PROPERTY P_scFuse_fbxEnable : CtaSysConfig.ITF_DATATYPE
GET
END_GET
END_PROPERTY

PROPERTY P_scFuse_fbxInputMb : CtaSysConfig.ITF_DATATYPE
GET
END_GET
END_PROPERTY

PROPERTY P_scFuse_fbxDoesAlarm : CtaSysConfig.ITF_DATATYPE
GET
END_GET
END_PROPERTY

PROPERTY P_scMotorFuse_fbxInputMb : CtaSysConfig.ITF_DATATYPE
GET
END_GET
END_PROPERTY

PROPERTY P_scMotorFuse_fbxEnable : CtaSysConfig.ITF_DATATYPE
GET
END_GET
END_PROPERTY

PROPERTY P_scMotorFuse_fbxDoesAlarm : CtaSysConfig.ITF_DATATYPE
GET
END_GET
END_PROPERTY

PROPERTY P_scManual_fbxAlowManualOn : CtaSysConfig.ITF_DATATYPE
GET
END_GET
END_PROPERTY

PROPERTY P_scManual_fbuiManualState : CtaSysConfig.ITF_DATATYPE
GET
END_GET
END_PROPERTY

PROPERTY P_scManual_fbrManualOnY : CtaSysConfig.ITF_DATATYPE
GET
END_GET
END_PROPERTY

PROPERTY P_scInfluxDb_fbxEnable : CtaSysConfig.ITF_DATATYPE
GET
END_GET
END_PROPERTY

PROPERTY P_scData_fbudiOperationStarts : CtaSysConfig.ITF_DATATYPE
GET
END_GET
END_PROPERTY

PROPERTY P_scData_fbudiOperatingHours : CtaSysConfig.ITF_DATATYPE
GET
END_GET
END_PROPERTY

PROPERTY proRefToRonYDumper : REFERENCE TO CtaAppDumper.fbDumper
GET
END_GET
END_PROPERTY

{attribute 'hide'} 
PROPERTY INTERNAL proCountedError : INT
GET
END_GET
END_PROPERTY

{attribute 'hide'} 
PROPERTY INTERNAL proCountedInfo : INT
GET
END_GET
END_PROPERTY

{attribute 'hide'} 
PROPERTY INTERNAL proITF_REPORTMANAGER : CtaAppReport.ITF_REPORTMANAGER
GET
END_GET
END_PROPERTY

{attribute 'hide'} 
PROPERTY INTERNAL proCountedWarning : INT
GET
END_GET
END_PROPERTY

PROPERTY INTERNAL proGetDI_MotorHand : BOOL
GET
END_GET
END_PROPERTY

{attribute 'hide'} 
PROPERTY proNotShowDI_MotorHand : BOOL
GET
END_GET
END_PROPERTY

PROPERTY proHandModul_ITF : CtaSysIO.ITF_IO
GET
END_GET
END_PROPERTY

PROPERTY proNotShowAI_ActualValue : BOOL
GET
END_GET
END_PROPERTY

PROPERTY proGetAI_ActualValue : REAL
GET
END_GET
END_PROPERTY

PROPERTY proActualValue_ITF : CtaSysIO.ITF_IO
GET
END_GET
END_PROPERTY

{attribute 'hide'} 
PROPERTY proNotShowDI_NoError : BOOL
GET
END_GET
END_PROPERTY

PROPERTY INTERNAL proGetDI_NoError : BOOL
GET
END_GET
END_PROPERTY

PROPERTY proNoError_ITF : CtaSysIO.ITF_IO
GET
END_GET
END_PROPERTY

{attribute 'hide'} 
PROPERTY proNotShowDI_RevisionSwitchOk : BOOL
GET
END_GET
END_PROPERTY

PROPERTY INTERNAL proGetDI_RevisionSwitchOK : BOOL
GET
END_GET
END_PROPERTY

PROPERTY proRevisionSwitch_ITF : CtaSysIO.ITF_IO
GET
END_GET
END_PROPERTY

{attribute 'hide'} 
PROPERTY proNotShowDI_IsOn : BOOL
GET
END_GET
END_PROPERTY

PROPERTY INTERNAL proGetDI_IsOn : BOOL
GET
END_GET
END_PROPERTY

PROPERTY proIsOn_ITF : CtaSysIO.ITF_IO
GET
END_GET
END_PROPERTY

{attribute 'hide'} 
PROPERTY proNotShowDI_MotorFuseOk : BOOL
GET
END_GET
END_PROPERTY

PROPERTY INTERNAL proGetDI_MotorFuseOk : BOOL
GET
END_GET
END_PROPERTY

PROPERTY proMotorFuse_ITF : CtaSysIO.ITF_IO
GET
END_GET
END_PROPERTY

{attribute 'hide'} 
PROPERTY proNotShowDI_FuseOk : BOOL
GET
END_GET
END_PROPERTY

PROPERTY INTERNAL proGetDI_FuseOK : BOOL
GET
END_GET
END_PROPERTY

PROPERTY proFuse_ITF : CtaSysIO.ITF_IO
GET
END_GET
END_PROPERTY

{attribute 'hide'} 
PROPERTY proNotShowDI_Ready : BOOL
GET
END_GET
END_PROPERTY

PROPERTY INTERNAL proGetDI_IsReady : BOOL
GET
END_GET
END_PROPERTY

PROPERTY proReady_ITF : CtaSysIO.ITF_IO
GET
END_GET
END_PROPERTY

PROPERTY proOn_ITF : CtaSysIO.ITF_IO
GET
END_GET
END_PROPERTY

PROPERTY proOnY_ITF : CtaSysIO.ITF_IO
GET
END_GET
END_PROPERTY

PROPERTY proIsRegulatet : BOOL
GET
END_GET
END_PROPERTY

PROPERTY proIsHandOnOrOff : BOOL
GET
END_GET
END_PROPERTY

PROPERTY proRunAfterTimeAktive : BOOL
GET
END_GET
END_PROPERTY

PROPERTY proLeadTimeAktive : BOOL
GET
END_GET
END_PROPERTY

PROPERTY proIsReady : BOOL
GET
END_GET
END_PROPERTY

PROPERTY proAuto : BOOL
GET
END_GET
SET
END_SET
END_PROPERTY

PROPERTY proHandOn : BOOL
SET
END_SET
GET
END_GET
END_PROPERTY

PROPERTY proIsError : BOOL
GET
END_GET
END_PROPERTY

PROPERTY proIsWarning : BOOL
GET
END_GET
END_PROPERTY

PROPERTY proEn : BOOL
GET
END_GET
SET
END_SET
END_PROPERTY

PROPERTY proHardWareHandModulAktive : BOOL
GET
END_GET
END_PROPERTY

PROPERTY proIsEnabled : BOOL
GET
END_GET
END_PROPERTY

PROPERTY proMotorIsOn : BOOL
GET
END_GET
END_PROPERTY

PROPERTY proHandOff : BOOL
SET
END_SET
GET
END_GET
END_PROPERTY

PROPERTY proRevisionSwitchOk : BOOL
GET
END_GET
END_PROPERTY

PROPERTY proHandOnY : REAL
SET
END_SET
GET
END_GET
END_PROPERTY

{attribute 'monitoring' := 'variable'}
PROPERTY proLockDown : BOOL
GET
END_GET
END_PROPERTY

{attribute 'monitoring' := 'variable'}
PROPERTY proAvailable : BOOL
GET
END_GET
END_PROPERTY

{attribute 'monitoring' := 'variable'}
PROPERTY proAcknowlege : BOOL
GET
END_GET
END_PROPERTY

PROPERTY proIconNr : UINT
SET
END_SET
GET
END_GET
END_PROPERTY

END_INTERFACE

// 30 Program Organization Units/fbAntrieb_Collector
FUNCTION_BLOCK fbAntrieb_Collector IMPLEMENTS ITF_ANTRIEB_COLLECTOR
VAR_INPUT
END_VAR
VAR_OUTPUT
END_VAR
VAR
    ayAT_INTERFACE          : ARRAY[1..Parameter.iMaxAT] OF ITF_ANTRIEB;   
    ayAT_INTERFACE_SORTET   : ARRAY[1..Parameter.iMaxAT] OF ITF_ANTRIEB; 
    xIsSortet               : BOOL;
    diNext                  : DINT    := 1;
    diMin                   : DINT    := 1;
    diMax                   : DINT;
    diMaxSort               : DINT;
    xError                  : BOOL;
    xBufferError            : BOOL;
    diMissedBuffer          : DINT;
END_VAR

METHOD metRegistry : DINT
VAR_INPUT
    ITF_AT_IN   :   ITF_ANTRIEB;
END_VAR
VAR
    diArrayPos  :   DINT;
    diCount     :   DINT;
END_VAR
IF ITF_AT_IN <> 0 THEN
    diArrayPos := __XADD(ADR(diNext),1);
    IF diArrayPos <= Parameter.iMaxAT AND diArrayPos >= 1 THEN
        IF __QUERYINTERFACE(ITF_AT_IN,ayAT_INTERFACE[diArrayPos]) THEN
            metRegistry             := diArrayPos;
            GVL_ANTRIEB.xValidData       := TRUE;
            diCount    := __XADD(ADR(diMax),1);
        END_IF;
    ELSE
        IF diArrayPos > Parameter.iMaxAT THEN
            xBufferError := TRUE;
            diMissedBuffer := diArrayPos - Parameter.iMaxAT;
		END_IF;
        xError      := TRUE; 
        metRegistry := 0;
    END_IF;   
ELSE
    xError := TRUE; 
    metRegistry := 0;
END_IF;
END_METHOD

METHOD metSortArray
VAR_INPUT
    stSearch    :   STRING;
    uiSort      :   UINT;
END_VAR
VAR
    diFor1      :   DINT;
    diFor2      :   DINT;
    diFill      :   DINT;
    ITF_AT_Temp :   ITF_ANTRIEB;    
    iBigger     :   INT;
END_VAR
IF stSearch <> '' THEN
    diMaxSort   := 0;
    diFill      := LOWER_BOUND(ayAT_INTERFACE,1); 
    FOR diFor1 := LOWER_BOUND(ayAT_INTERFACE,1) TO UPPER_BOUND(ayAT_INTERFACE,1) DO
        IF ayAT_INTERFACE[diFor1] <> 0 THEN
            IF FIND(ayAT_INTERFACE[diFor1].proGetBMK,stSearch) <> 0 OR FIND(ayAT_INTERFACE[diFor1].proGetVendorDesignation,stSearch) <> 0 THEN
                ayAT_INTERFACE_SORTET[diFill] := ayAT_INTERFACE[diFor1];
                diFill      := diFill + 1; 
                diMaxSort   := diFill -1; 
            END_IF;
        END_IF;
	END_FOR;
ELSE
    ayAT_INTERFACE_SORTET := ayAT_INTERFACE;
    diMaxSort := diMax;
END_IF; 
// 1 = Sort BMK
IF uiSort = 1 THEN
    FOR diFor1 := LOWER_BOUND(ayAT_INTERFACE_SORTET,1) TO diMaxSort DO 
        FOR diFor2 := LOWER_BOUND(ayAT_INTERFACE_SORTET,1) TO diMaxSort -1 DO 
            IF ayAT_INTERFACE_SORTET[diFor2] <> 0 AND ayAT_INTERFACE_SORTET[diFor2 + 1] <> 0 THEN
                IF LEN(ayAT_INTERFACE_SORTET[diFor2].proGetBMK) > LEN(ayAT_INTERFACE_SORTET[diFor2 + 1].proGetBMK) THEN
                    ITF_AT_Temp                         := ayAT_INTERFACE_SORTET[diFor2];
                    ayAT_INTERFACE_SORTET[diFor2]       := ayAT_INTERFACE_SORTET[diFor2 + 1];
                    ayAT_INTERFACE_SORTET[diFor2 + 1]   := ITF_AT_Temp; 
                ELSIF LEN(ayAT_INTERFACE_SORTET[diFor2].proGetBMK) = LEN(ayAT_INTERFACE_SORTET[diFor2 + 1].proGetBMK) THEN
                    iBigger := fcGetBigerStringValue(ayAT_INTERFACE_SORTET[diFor2].proGetBMK,ayAT_INTERFACE_SORTET[diFor2 + 1].proGetBMK);
                    IF iBigger = 1 THEN
                        ITF_AT_Temp                         := ayAT_INTERFACE_SORTET[diFor2];
                        ayAT_INTERFACE_SORTET[diFor2]       := ayAT_INTERFACE_SORTET[diFor2 + 1];
                        ayAT_INTERFACE_SORTET[diFor2 + 1]   := ITF_AT_Temp;                                                
					END_IF;
				END_IF;
            END_IF;       
        END_FOR;      
    END_FOR;     
// 2 = Sort Vendor Name    
ELSIF uiSort = 2 THEN
    FOR diFor1 := LOWER_BOUND(ayAT_INTERFACE_SORTET,1) TO diMaxSort DO 
        FOR diFor2 := LOWER_BOUND(ayAT_INTERFACE_SORTET,1) TO diMaxSort -1 DO 
            IF ayAT_INTERFACE_SORTET[diFor2] <> 0 AND ayAT_INTERFACE_SORTET[diFor2 + 1] <> 0 THEN
                iBigger := fcGetBigerStringValue(ayAT_INTERFACE_SORTET[diFor2].proGetVendorDesignation,ayAT_INTERFACE_SORTET[diFor2 + 1].proGetVendorDesignation);
                IF iBigger = 1 THEN
                    ITF_AT_Temp                         := ayAT_INTERFACE_SORTET[diFor2];
                    ayAT_INTERFACE_SORTET[diFor2]       := ayAT_INTERFACE_SORTET[diFor2 + 1];
                    ayAT_INTERFACE_SORTET[diFor2 + 1]   := ITF_AT_Temp;                                            
                END_IF;
            END_IF;       
        END_FOR;      
    END_FOR;
// 3 & 4 = Sort State  
ELSIF uiSort = 3 OR uiSort = 4 THEN
    FOR diFor1 := LOWER_BOUND(ayAT_INTERFACE_SORTET,1) TO diMaxSort DO 
        FOR diFor2 := LOWER_BOUND(ayAT_INTERFACE_SORTET,1) TO diMaxSort -1 DO 
            IF ayAT_INTERFACE_SORTET[diFor2] <> 0 AND ayAT_INTERFACE_SORTET[diFor2 + 1] <> 0 THEN
                IF ayAT_INTERFACE_SORTET[diFor2].proIsError < ayAT_INTERFACE_SORTET[diFor2 + 1].proIsError THEN
                    ITF_AT_Temp                         := ayAT_INTERFACE_SORTET[diFor2];
                    ayAT_INTERFACE_SORTET[diFor2]       := ayAT_INTERFACE_SORTET[diFor2 + 1];
                    ayAT_INTERFACE_SORTET[diFor2 + 1]   := ITF_AT_Temp;    
                ELSIF NOT ayAT_INTERFACE_SORTET[diFor2].proIsError THEN
                    IF ayAT_INTERFACE_SORTET[diFor2].proIsWarning < ayAT_INTERFACE_SORTET[diFor2 + 1].proIsWarning THEN
                        ITF_AT_Temp                         := ayAT_INTERFACE_SORTET[diFor2];
                        ayAT_INTERFACE_SORTET[diFor2]       := ayAT_INTERFACE_SORTET[diFor2 + 1];
                        ayAT_INTERFACE_SORTET[diFor2 + 1]   := ITF_AT_Temp;    
                    ELSIF ayAT_INTERFACE_SORTET[diFor2].proIsEnabled < ayAT_INTERFACE_SORTET[diFor2 + 1].proIsEnabled THEN
                        ITF_AT_Temp                         := ayAT_INTERFACE_SORTET[diFor2];
                        ayAT_INTERFACE_SORTET[diFor2]       := ayAT_INTERFACE_SORTET[diFor2 + 1];
                        ayAT_INTERFACE_SORTET[diFor2 + 1]   := ITF_AT_Temp; 
                    ELSIF ayAT_INTERFACE_SORTET[diFor2].proIsWarning AND ayAT_INTERFACE_SORTET[diFor2 + 1].proIsWarning THEN
                        IF ayAT_INTERFACE_SORTET[diFor2].proRevisionSwitchOk > ayAT_INTERFACE_SORTET[diFor2 + 1].proRevisionSwitchOk THEN         
                            ITF_AT_Temp                         := ayAT_INTERFACE_SORTET[diFor2];
                            ayAT_INTERFACE_SORTET[diFor2]       := ayAT_INTERFACE_SORTET[diFor2 + 1];
                            ayAT_INTERFACE_SORTET[diFor2 + 1]   := ITF_AT_Temp; 
                        END_IF;       
                    END_IF;                                                       
                END_IF;
            END_IF;       
        END_FOR;      
    END_FOR;    
// 5 = Sort Starts   
ELSIF uiSort = 5 THEN
    FOR diFor1 := LOWER_BOUND(ayAT_INTERFACE_SORTET,1) TO diMaxSort DO 
        FOR diFor2 := LOWER_BOUND(ayAT_INTERFACE_SORTET,1) TO diMaxSort -1 DO 
            IF ayAT_INTERFACE_SORTET[diFor2] <> 0 AND ayAT_INTERFACE_SORTET[diFor2 + 1] <> 0 THEN
                IF ayAT_INTERFACE_SORTET[diFor2].proCountedStarts < ayAT_INTERFACE_SORTET[diFor2 + 1].proCountedStarts THEN
                    ITF_AT_Temp                         := ayAT_INTERFACE_SORTET[diFor2];
                    ayAT_INTERFACE_SORTET[diFor2]       := ayAT_INTERFACE_SORTET[diFor2 + 1];
                    ayAT_INTERFACE_SORTET[diFor2 + 1]   := ITF_AT_Temp;                                            
                END_IF;
            END_IF;       
        END_FOR;      
    END_FOR; 
// 6 = Sort Stunden   
ELSIF uiSort = 6 THEN
    FOR diFor1 := LOWER_BOUND(ayAT_INTERFACE_SORTET,1) TO diMaxSort DO 
        FOR diFor2 := LOWER_BOUND(ayAT_INTERFACE_SORTET,1) TO diMaxSort -1 DO 
            IF ayAT_INTERFACE_SORTET[diFor2] <> 0 AND ayAT_INTERFACE_SORTET[diFor2 + 1] <> 0 THEN
                IF ayAT_INTERFACE_SORTET[diFor2].proCountedHours < ayAT_INTERFACE_SORTET[diFor2 + 1].proCountedHours THEN
                    ITF_AT_Temp                         := ayAT_INTERFACE_SORTET[diFor2];
                    ayAT_INTERFACE_SORTET[diFor2]       := ayAT_INTERFACE_SORTET[diFor2 + 1];
                    ayAT_INTERFACE_SORTET[diFor2 + 1]   := ITF_AT_Temp;                                            
                END_IF;
            END_IF;       
        END_FOR;      
    END_FOR;   
// 7 = Sort On   
ELSIF uiSort = 7 THEN
    FOR diFor1 := LOWER_BOUND(ayAT_INTERFACE_SORTET,1) TO diMaxSort DO 
        FOR diFor2 := LOWER_BOUND(ayAT_INTERFACE_SORTET,1) TO diMaxSort -1 DO 
            IF ayAT_INTERFACE_SORTET[diFor2] <> 0 AND ayAT_INTERFACE_SORTET[diFor2 + 1] <> 0 THEN
                IF ayAT_INTERFACE_SORTET[diFor2].proOn < ayAT_INTERFACE_SORTET[diFor2 + 1].proOn THEN
                    ITF_AT_Temp                         := ayAT_INTERFACE_SORTET[diFor2];
                    ayAT_INTERFACE_SORTET[diFor2]       := ayAT_INTERFACE_SORTET[diFor2 + 1];
                    ayAT_INTERFACE_SORTET[diFor2 + 1]   := ITF_AT_Temp;                                            
                END_IF;
            END_IF;       
        END_FOR;      
    END_FOR;   
ELSE
    uiSort := 0;     
END_IF; 
IF uiSort = 0 AND stSearch = '' THEN
    xIsSortet := FALSE;  
ELSE
    xIsSortet := TRUE;  
END_IF
END_METHOD

PROPERTY proMin : INT
GET
proMin := 1;
END_GET
END_PROPERTY

PROPERTY proMax : UINT
GET
IF xIsSortet THEN
    proMax := LIMIT(0,TO_UINT(diMaxSort),65535);    
ELSE
    proMax := LIMIT(0,TO_UINT(diMax),65535);    
END_IF
END_GET
END_PROPERTY

PROPERTY proayAntriebTabelle : ARRAY[1..Parameter.iMaxAT] OF ITF_ANTRIEB_TABELLE_INFO
GET
VAR
    diFor   :   DINT;
END_VAR
IF xIsSortet THEN
    FOR diFor := LOWER_BOUND(proayAntriebTabelle,1) TO UPPER_BOUND(proayAntriebTabelle,1) DO
        __QUERYINTERFACE(ayAT_INTERFACE_SORTET[diFor],proayAntriebTabelle[diFor]);   
	END_FOR
ELSE
    FOR diFor := LOWER_BOUND(proayAntriebTabelle,1) TO UPPER_BOUND(proayAntriebTabelle,1) DO
        __QUERYINTERFACE(ayAT_INTERFACE[diFor],proayAntriebTabelle[diFor]);   
	END_FOR
END_IF;
END_GET
END_PROPERTY

PROPERTY proMissedBuffer : DINT
GET
proMissedBuffer := diMissedBuffer;
END_GET
END_PROPERTY

PROPERTY proBufferError : BOOL
GET
proBufferError := xBufferError;
END_GET
END_PROPERTY

PROPERTY proayAntrieb : ARRAY[1..Parameter.iMaxAT] OF ITF_ANTRIEB
GET
VAR
    diFor   :   DINT;
END_VAR
IF xIsSortet THEN
    proayAntrieb := ayAT_INTERFACE_SORTET;
ELSE
    proayAntrieb := ayAT_INTERFACE;
END_IF;
END_GET
END_PROPERTY

METHOD metGetAntriebITF : ITF_ANTRIEB
VAR_INPUT
    iPos    :   INT;
END_VAR
IF TO_DINT(iPos) >= LOWER_BOUND(ayAT_INTERFACE,1) AND TO_DINT(iPos) <= UPPER_BOUND(ayAT_INTERFACE,1) THEN
    IF xIsSortet THEN
        metGetAntriebITF := ayAT_INTERFACE_SORTET[iPos];       
    ELSE
        metGetAntriebITF := ayAT_INTERFACE[iPos];       
	END_IF   
END_IF
END_METHOD

END_FUNCTION_BLOCK

// 21 Interface/ITF_ANTRIEB_COLLECTOR
INTERFACE ITF_ANTRIEB_COLLECTOR

PROPERTY proBufferError : BOOL
GET
END_GET
END_PROPERTY

METHOD metGetAntriebITF : ITF_ANTRIEB
VAR_INPUT
    iPos    :   INT;
END_VAR
END_METHOD

PROPERTY proMissedBuffer : DINT
GET
END_GET
END_PROPERTY

PROPERTY proMin : INT
GET
END_GET
END_PROPERTY

PROPERTY proMax : UINT
GET
END_GET
END_PROPERTY

PROPERTY proayAntriebTabelle : ARRAY[1..Parameter.iMaxAT] OF ITF_ANTRIEB_TABELLE_INFO
GET
END_GET
END_PROPERTY

METHOD metSortArray
VAR_INPUT
    stSearch    :   STRING;
    uiSort      :   UINT;
END_VAR
END_METHOD

END_INTERFACE

// 30 Program Organization Units/fcGetBigerStringValue
FUNCTION fcGetBigerStringValue : INT
VAR_INPUT
    st1     :   STRING(255);
    st2     :   STRING(255);
END_VAR
VAR
    diFor: DINT;
    diMax: DINT;
END_VAR

IF LEN(st1) > LEN(st2) THEN
    diMax := LEN(st2); 
    fcGetBigerStringValue := 1;
ELSIF LEN(st1) < LEN(st2) THEN
    diMax := LEN(st1);
    fcGetBigerStringValue := 2;     
ELSE
    diMax := LEN(st1);    
END_IF;
FOR diFor := 0 TO  diMax DO
    IF st1[diFor] > st2[diFor] THEN
        fcGetBigerStringValue := 1;  
        EXIT; 
    ELSIF st1[diFor] < st2[diFor] THEN
        fcGetBigerStringValue := 2;  
        EXIT;
    END_IF;
END_FOR;

END_FUNCTION

// 30 Program Organization Units/fcCheckQuerryAndIconReturn
FUNCTION fcCheckQuerryAndIconReturn : BOOL
VAR_INPUT
	_ITF_IN			: 	ITF_ANTRIEB;
	_uiIconNr_IN	:	UINT;
END_VAR

IF __QUERYINTERFACE(_ITF_IN,_ITF_IN) THEN
	fcCheckQuerryAndIconReturn := TRUE;	
	_ITF_IN.proIconNr := _uiIconNr_IN;
ELSE
	fcCheckQuerryAndIconReturn :=  FALSE;
END_IF

END_FUNCTION

// 40 Visualizations/COLLECTOR/VIS_ANTRIEB_COLLECTOR
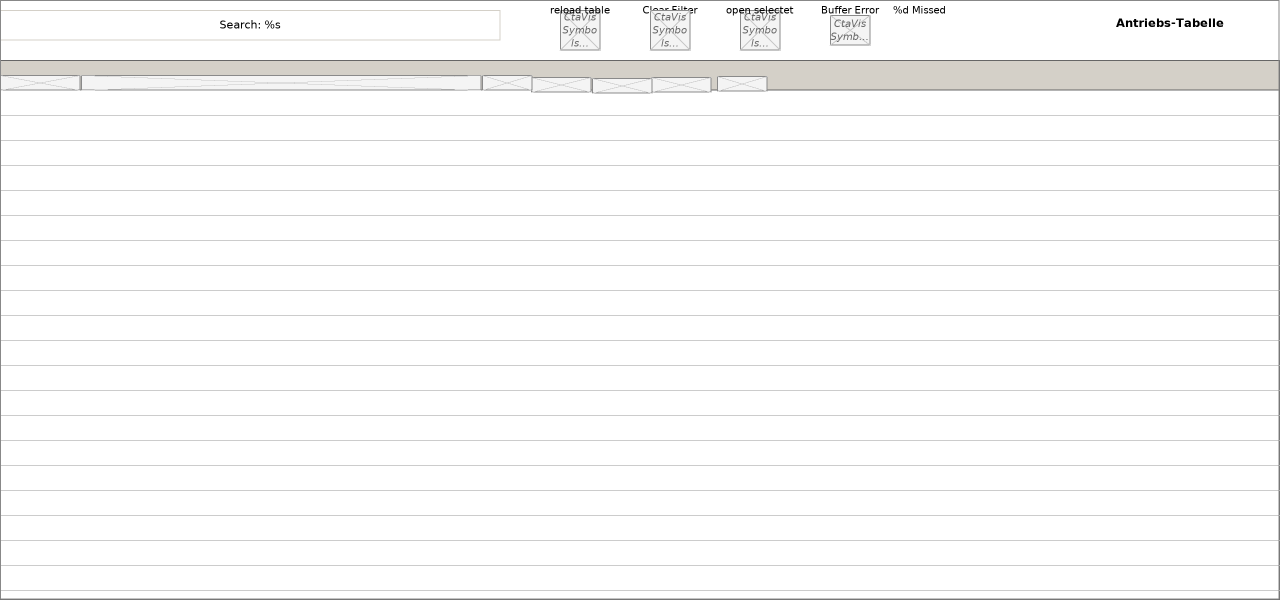
VISUALIZATION VIS_ANTRIEB_COLLECTOR  // 1280x600
    Frame (0,0 1280x600), invisible if: NOT GVL_ANTRIEB.xValidData
        shows VIS_ANTRIEB_COLLECTOR_TEMP(ayAntriebTabellenInfo := GVL_ANTRIEB.fbAntrieb_Collector.proayAntriebTabelle, uiMax := GVL_ANTRIEB.fbAntrieb_Collector.proMax, ITF_ANTRIEB_COLLECTOR := GVL_ANTRIEB.fbAntrieb_Collector)
END_VISUALIZATION

// 40 Visualizations/COLLECTOR/Help Funktionen/SelSort
VISUALIZATION SelSort  // 15x30
VAR_IN_OUT
	uiSel                       :   UINT;
END_VAR
VAR_INPUT
    stSearch                    :   STRING;    
    ITF_ANTRIEB_COLLECTOR       : ITF_ANTRIEB_COLLECTOR;
END_VAR
VAR_INPUT CONSTANT
    uiValue             :   UINT;
END_VAR
    Frame (0,15 15x15), invisible if: uiValue <> uiSel
        shows SortPfeil()
    Rectangle (0,0 15x30)
        OnMouseClick: execute {
            IF uiSel <> uiValue THEN
                uiSel   := uiValue;
            ELSE
                uiSel   := 0;
            END_IF
            ITF_ANTRIEB_COLLECTOR.metSortArray(stSearch,uiSel);
        }
END_VISUALIZATION

// 40 Visualizations/COLLECTOR/VIS_ANTRIEB_COLLECTOR_TEMP
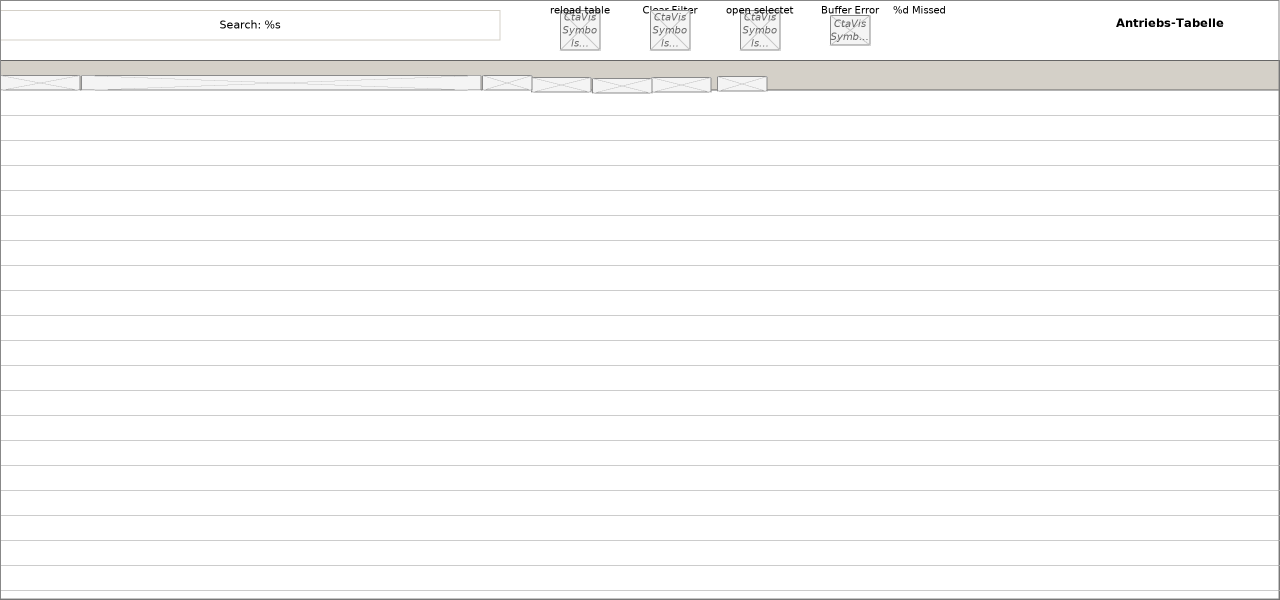
VISUALIZATION VIS_ANTRIEB_COLLECTOR_TEMP  // 1280x600
VAR_INPUT
	ayAntriebTabellenInfo   : ARRAY[1..Parameter.iMaxAT] OF ITF_ANTRIEB_TABELLE_INFO;
    uiMax                   : UINT;
    ITF_ANTRIEB_COLLECTOR   : ITF_ANTRIEB_COLLECTOR;
END_VAR
VAR
    iZeile                  :   INT;
    stSearch                :   STRING;
    uiSort                  :   UINT;
    xReadySearch            :   BOOL;
END_VAR
    Table (0,60 1280x540), data array: ayAntriebTabellenInfo
        p1128707560: uiMax
        p1014161805: Parameter.iMaxAT - 1 + 1
        p1137915858: iZeile
        p3726181087: ayAntriebTabellenInfo[INDEX].proNoBmkInList
        p3136911649: ayAntriebTabellenInfo[INDEX].proGetInstancePath
        p797552052: ayAntriebTabellenInfo[INDEX].proSetInstancePath
        p3854506369: ayAntriebTabellenInfo[INDEX].proGetBMK
        p1744040210: ayAntriebTabellenInfo[INDEX].proGetObjectId
        p290089404: ayAntriebTabellenInfo[INDEX].proGetCustomerDesignation
        p2319025000: ayAntriebTabellenInfo[INDEX].proGetAKS
        p511219082: Vendor designation
        p1892666644: ayAntriebTabellenInfo[INDEX].proGetVendorDesignation
        p4242324053: Run-on time
        p3863566920: ayAntriebTabellenInfo[INDEX].proRunAfterTime
        p1755163831: State
        p338671338: ayAntriebTabellenInfo[INDEX].proStateSymbol
        p505689113: Hours
        p1218418051: ayAntriebTabellenInfo[INDEX].proCountedHours
        p2340480326: ayAntriebTabellenInfo[INDEX].proBetriebsstunden
        p2237128397: Starts
        p3723444502: ayAntriebTabellenInfo[INDEX].proCountedStarts
        p4008173056: ayAntriebTabellenInfo[INDEX].proAnzahlStarts
        p4092479075: Enabled
        p2170511999: ayAntriebTabellenInfo[INDEX].proEnSymbol
        p4088588272: On IN
        p3104783080: ayAntriebTabellenInfo[INDEX].proIsOn
        p1757482276: On OUT
        p746581629: ayAntriebTabellenInfo[INDEX].proOn
        p1739542657: Lead time
        p1933151965: ayAntriebTabellenInfo[INDEX].proLeadTime
        p516019884: Y IN
        p7306298: ayAntriebTabellenInfo[INDEX].proIsOnY
        p2243050616: Y OUT
        p2501879983: ayAntriebTabellenInfo[INDEX].proOnY
    Image (740,10 40x40), invisible if: TO_DINT(iZeile) < LOWER_BOUND(ayAntriebTabellenInfo,1) OR TO_DINT(iZeile) > UPPER_BOUND(ayAntriebTabellenInfo,1), image: CtaVisSymbols.ImagePool.engine
        OnMouseClick:  Dialog=POPUP_ANTRIEB, Parameters={ITF_ANTRIEBIN: ITF_ANTRIEB_COLLECTOR.metGetAntriebITF(iZeile), uiPopUpGruppe: 0}, OpenModal=True, OpenCentered=True
    Textfield (0,10 500x30), "Search: %s", text variable: stSearch
        OnMouseClick: write the text variable via Default
        OnMouseClick: execute { xReadySearch := TRUE; }
    Image (560,10 40x40), invisible if: NOT xReadySearch, image: CtaVisSymbols.ImagePool.refresh_solo_black
        OnMouseClick: execute { ITF_ANTRIEB_COLLECTOR.metSortArray(stSearch,uiSort); xReadySearch := FALSE; }
    Label (540,5 80x10), "reload table", invisible if: NOT xReadySearch
    Label (720,5 80x10), "open selectet", invisible if: TO_DINT(iZeile) < LOWER_BOUND(ayAntriebTabellenInfo,1) OR TO_DINT(iZeile) > UPPER_BOUND(ayAntriebTabellenInfo,1)
    Label (630,5 80x10), "Clear Filter", invisible if: stSearch = '' AND uiSort = 0
    Image (650,10 40x40), invisible if: stSearch = '' AND uiSort = 0, image: CtaVisSymbols.ImagePool.close_solo_black
        OnMouseClick: execute {
            stSearch := '';
            uiSort   := 0;
            ITF_ANTRIEB_COLLECTOR.metSortArray(stSearch,uiSort);
            xReadySearch := FALSE;
        }
    Label (1095,8 150x30), "Antriebs-Tabelle"
    Label (810,5 80x10), "Buffer Error", invisible if: NOT ITF_ANTRIEB_COLLECTOR.proBufferError
    Image (830,15 40x30), invisible if: NOT ITF_ANTRIEB_COLLECTOR.proBufferError, image: CtaVisSymbols.ImagePool.CtaError
    Textfield (890,5 100x10), "%d Missed", text variable: ITF_ANTRIEB_COLLECTOR.proMissedBuffer, invisible if: NOT ITF_ANTRIEB_COLLECTOR.proBufferError
    Frame (717,61 50x30)
        shows SelSort(uiSel := uiSort, stSearch := stSearch, ITF_ANTRIEB_COLLECTOR := ITF_ANTRIEB_COLLECTOR, uiValue := 7)
    Frame (651,62 60x30)
        shows SelSort(uiSel := uiSort, stSearch := stSearch, ITF_ANTRIEB_COLLECTOR := ITF_ANTRIEB_COLLECTOR, uiValue := 6)
    Frame (592,63 60x30)
        shows SelSort(uiSel := uiSort, stSearch := stSearch, ITF_ANTRIEB_COLLECTOR := ITF_ANTRIEB_COLLECTOR, uiValue := 5)
    Frame (531,62 60x30)
        shows SelSort(uiSel := uiSort, stSearch := stSearch, ITF_ANTRIEB_COLLECTOR := ITF_ANTRIEB_COLLECTOR, uiValue := 4)
    Frame (482,60 50x30)
        shows SelSort(uiSel := uiSort, stSearch := stSearch, ITF_ANTRIEB_COLLECTOR := ITF_ANTRIEB_COLLECTOR, uiValue := 3)
    Frame (81,60 400x30)
        shows SelSort(uiSel := uiSort, stSearch := stSearch, ITF_ANTRIEB_COLLECTOR := ITF_ANTRIEB_COLLECTOR, uiValue := 2)
    Frame (0,60 80x30)
        shows SelSort(uiSel := uiSort, stSearch := stSearch, ITF_ANTRIEB_COLLECTOR := ITF_ANTRIEB_COLLECTOR, uiValue := 1)
END_VISUALIZATION

// 40 Visualizations/COLLECTOR/Help Funktionen/SortPfeil
VISUALIZATION SortPfeil  // 15x15
    Image (0,0 15x15), image: CtaVisSymbols.ImagePool.arrow-down_solo_black
END_VISUALIZATION

// 40 Visualizations/POPUP/POPUP_ANTRIEB
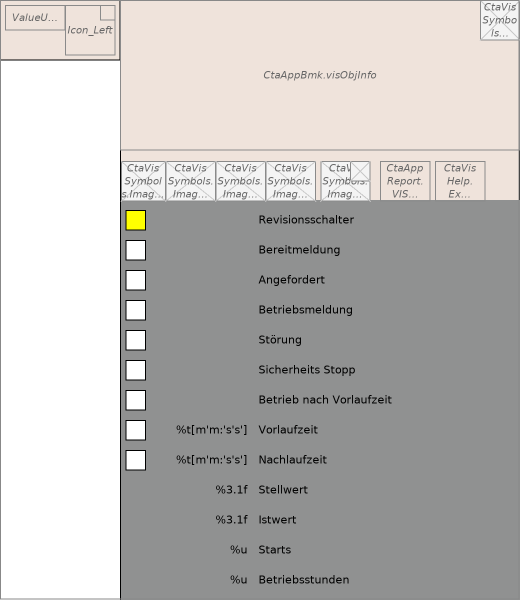
VISUALIZATION POPUP_ANTRIEB  // 520x600
VAR_INPUT
    ITF_ANTRIEBIN    	:   ITF_ANTRIEB;
	stExklParameter_IN	:	STRING[40];	
	uiPopUpGruppe 		: 	UINT;
END_VAR
    Rectangle (0,0 120x60)
    Rectangle (120,0 400x600)
    Frame (120,0 400x150)
        shows CtaAppBmk.visObjInfo(ITF_BMK_IN := ITF_ANTRIEBIN)
    Image (480,0 40x40), image: CtaVisSymbols.ImagePool.close_solo_black
        OnMouseClick:  Dialog=POPUP_ANTRIEB, Result=None, NumpadKeypadSet=True
    Frame (121,200 399x400), frame switch variable: uiPopUpGruppe
        shows VIS_ANTRIEB_OVERVIEW(ITF_ANTRIEBIN := ITF_ANTRIEBIN)
        shows VIS_ANTRIEB_MANUAL(ITF_ANTRIEBIN := ITF_ANTRIEBIN)
        shows VIS_ANTRIEB_PARAMETER(ITF_ANTRIEBIN := ITF_ANTRIEBIN)
        shows VIS_ANTRIEB_IO(ITF_ANTRIEBIN := ITF_ANTRIEBIN)
        shows AT_BUS(ITF_ANTRIEBIN := ITF_ANTRIEBIN)
        shows VIS_ANTRIEB_REPORTS(ITF_ANTRIEBIN := ITF_ANTRIEBIN)
        pReferences[2]: ITF_Parameter=ITF_ANTRIEBIN.proParameter
    Frame (121,161 399x40)
        shows VIS_ANTRIEB_LISTE(uiPopUpGruppe := uiPopUpGruppe, xHand := ITF_ANTRIEBIN.proIsHandOnOrOff, xHandOff := ITF_ANTRIEBIN.proHandOff, ITF_REPORTMANAGER_IN := ITF_ANTRIEBIN.proITF_REPORTMANAGER, xBusTestAktiv := ITF_ANTRIEBIN.proModbusTest, stExklParameter_IN := stExklParameter_IN)
    Frame (5,5 110x50), input disabled if: TRUE, frame switch variable: ITF_ANTRIEBIN.proIconNr
        shows VIS_ANTRIEB_LEFT_ABOVE(ITF_ANTRIEB_IN := ITF_ANTRIEBIN, stExklParameter := stExklParameter_IN)
        shows VIS_ANTRIEB_LEFT_BELOW(ITF_ANTRIEB_IN := ITF_ANTRIEBIN, stExklParameter := stExklParameter_IN)
        shows VIS_ANTRIEB_RIGHT_ABOVE(ITF_ANTRIEB_IN := ITF_ANTRIEBIN, stExklParameter := stExklParameter_IN)
        shows VIS_ANTRIEB_RIGHT_BELOW(ITF_ANTRIEB_IN := ITF_ANTRIEBIN, stExklParameter := stExklParameter_IN)
END_VISUALIZATION

// 40 Visualizations/POPUP/VIS_ANTRIEB_LISTE
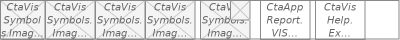
VISUALIZATION VIS_ANTRIEB_LISTE  // 400x40
VAR_IN_OUT
	uiPopUpGruppe 			:	UINT;
END_VAR
VAR_INPUT
    xHand           		: 	BOOL;
    xHandOff        		: 	BOOL;
    ITF_REPORTMANAGER_IN 	: 	CtaAppReport.ITF_REPORTMANAGER;
    xBusTestAktiv   		: 	BOOL;	
	stExklParameter_IN		:	STRING[40];
END_VAR
    Rectangle (100,0 40x40), colour toggle: uiPopUpGruppe = 2
        OnMouseDown: execute { uiPopUpGruppe := 2; }
    Rectangle (50,0 40x40), colour toggle: uiPopUpGruppe = 1
        OnMouseDown: execute { uiPopUpGruppe := 1; }
    Rectangle (0,0 40x40), colour toggle: uiPopUpGruppe = 0
        OnMouseDown: execute { uiPopUpGruppe := 0; }
    Image (0,0 45x40), image: CtaVisSymbols.ImagePool.eye
        OnMouseDown: execute { uiPopUpGruppe := 0; }
    Image (45,0 50x40), image: CtaVisSymbols.ImagePool.front_hand_Black
        OnMouseDown: execute { uiPopUpGruppe := 1; }
    Image (95,0 50x40), image: CtaVisSymbols.ImagePool.gear
        OnMouseDown: execute { uiPopUpGruppe := 2; }
    Image (45,0 50x40), invisible if: NOT xHand, image: CtaVisSymbols.ImagePool.front_hand_Yellow
        OnMouseDown: execute { uiPopUpGruppe := 1; }
    Rectangle (205,0 40x40), colour toggle: uiPopUpGruppe = 4
        OnMouseDown: execute { uiPopUpGruppe := 4; }
    Image (200,0 50x40), image: CtaVisSymbols.ImagePool.lan
        OnMouseDown: execute { uiPopUpGruppe := 4; }
    Image (45,0 50x40), invisible if: NOT xHandOff, image: CtaVisSymbols.ImagePool.front_hand_Yellow_Off
        OnMouseDown: execute { uiPopUpGruppe := 1; }
    Rectangle (150,0 40x40), colour toggle: uiPopUpGruppe = 3
        OnMouseDown: execute { uiPopUpGruppe := 3; }
    Image (145,0 50x40), image: CtaVisSymbols.ImagePool.dip-switch
        OnMouseDown: execute { uiPopUpGruppe := 3; }
    Image (230,0 20x20), invisible if: NOT xBusTestAktiv, image: CtaVisSymbols.ImagePool.front_hand_Yellow
        OnMouseDown: execute { uiPopUpGruppe := 4; }
    Rectangle (260,0 50x40), colour toggle: uiPopUpGruppe = 5
        OnMouseDown: execute { uiPopUpGruppe := 5; }
    Frame (260,0 50x40), input disabled if: TRUE
        shows CtaAppReport.VIS_ANZ_REPORTS_MODUL(ITF_REPORTMANAGER_IN := ITF_REPORTMANAGER_IN)
        OnMouseDown: execute { uiPopUpGruppe := 5; }
    Frame (315,0 50x40)
        shows CtaVisHelp.ExkParameterSymbol(stExklParameter := stExklParameter_IN)
END_VISUALIZATION

// 40 Visualizations/ICON/ANTRIEB_RIGHT/ANTRIEB_RIGHT_ABOVE/VIS_ANTRIEB_RigthAboveCheckQuerry
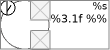
VISUALIZATION VIS_ANTRIEB_RigthAboveCheckQuerry  // 110x50
VAR_INPUT
    ITF_ANTRIEB_IN   :   ITF_ANTRIEB;	
END_VAR
VAR_INPUT
	stExklParameter		:	STRING[40];
END_VAR
    Frame (0,0 110x50)
        shows VIS_ANTRIEB_RigthAboveCheckIsEnabled(ITF_ANTRIEB_IN := ITF_ANTRIEB_IN, stExklParameter := stExklParameter)
END_VISUALIZATION

// 40 Visualizations/ICON/ANTRIEB_RIGHT/ANTRIEB_RIGHT_ABOVE/VIS_ANTRIEB_RIGHT_ABOVE
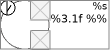
VISUALIZATION VIS_ANTRIEB_RIGHT_ABOVE  // 110x50
VAR_INPUT
    ITF_ANTRIEB_IN   :   ITF_ANTRIEB;	
END_VAR
VAR_INPUT CONSTANT
	stExklParameter		:	STRING[40] := ' ';
END_VAR
VAR CONSTANT
	uiIconNr		: UINT := 2;
END_VAR
    Frame (0,0 110x50), invisible if: NOT fcCheckQuerryAndIconReturn(_ITF_IN := ITF_ANTRIEB_IN, _uiIconNr_IN := uiIconNr)
        shows VIS_ANTRIEB_RigthAboveCheckQuerry(ITF_ANTRIEB_IN := ITF_ANTRIEB_IN, stExklParameter := stExklParameter)
END_VISUALIZATION

// 40 Visualizations/ICON/ANTRIEB_RIGHT/ANTRIEB_RIGHT_ABOVE/VIS_ANTRIEB_RigthAboveCheckIsEnabled
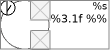
VISUALIZATION VIS_ANTRIEB_RigthAboveCheckIsEnabled  // 110x50
VAR_INPUT
    ITF_ANTRIEB_IN   :   ITF_ANTRIEB;	
END_VAR
VAR_INPUT
	stExklParameter		:	STRING[40];
END_VAR
    Frame (0,0 50x50), invisible if: NOT ITF_ANTRIEB_IN.proIsEnabled
        shows Icon_Right(ITF_ANTRIEB_IN := ITF_ANTRIEB_IN)
        shows Value_Right()
    Frame (50,0 60x25), invisible if: NOT ITF_ANTRIEB_IN.proIsEnabled
        shows ValueUpDwn(ITF_ANTRIEB_IN := ITF_ANTRIEB_IN, uiTextAusrichtung := 4)
    Frame (0,0 15x15), invisible if: NOT ITF_ANTRIEB_IN.proIsEnabled
        shows CommandOn(ITF_ANTRIEB_IN := ITF_ANTRIEB_IN)
    Rectangle (0,0 110x50)
        OnMouseClick:  Dialog=POPUP_ANTRIEB, Parameters={uiPopUpGruppe: 0, stExklParameter_IN: stExklParameter, ITF_ANTRIEBIN: ITF_ANTRIEB_IN}, OpenCentered=True
END_VISUALIZATION

// 40 Visualizations/ICON/ANTRIEB_BASE/CommandOn
VISUALIZATION CommandOn  // 15x15
VAR_INPUT
    ITF_ANTRIEB_IN   :   ITF_ANTRIEB;	
END_VAR
    Ellipse (0,0 15x15), colour toggle: ITF_ANTRIEB_IN.proOn
    Line (7,15) (7,10)
    Line (7,5) (7,0)
    Line (7,11) (11,5), invisible if: ITF_ANTRIEB_IN.proOn
    Line (7,15) (7,0), invisible if: NOT ITF_ANTRIEB_IN.proOn
END_VISUALIZATION

// 40 Visualizations/ICON/ANTRIEB_BASE/ICON/Icon_Left
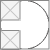
VISUALIZATION Icon_Left  // 50x50
VAR_INPUT
    ITF_ANTRIEB_IN   :   ITF_ANTRIEB;	
END_VAR
    Ellipse (0,0 49x49), colour toggle: ITF_ANTRIEB_IN.proMotorIsOn, invisible if: ITF_ANTRIEB_IN.proIsError
    Ellipse (0,0 49x49), colour toggle: ITF_ANTRIEB_IN.proIsError
    Image (0,0 20x20), invisible if: NOT ITF_ANTRIEB_IN.proIsWarning, image: CtaVisSymbols.ImagePool.CtaWarning
    Image (0,30 20x20), invisible if: NOT ITF_ANTRIEB_IN.proIsHandOnOrOff, image: CtaVisSymbols.ImagePool.front_hand_Yellow
    Image (0,30 20x20), invisible if: NOT ITF_ANTRIEB_IN.proHandOff, image: CtaVisSymbols.ImagePool.front_hand_Yellow_Off
END_VISUALIZATION

// 40 Visualizations/POPUP/PARAMETER/VIS_ANTRIEB_PARAMETER
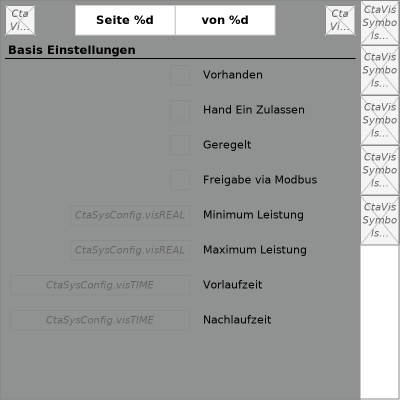
VISUALIZATION VIS_ANTRIEB_PARAMETER  // 400x400
VAR_INPUT
    ITF_ANTRIEBIN    :   ITF_ANTRIEB;	
END_VAR
VAR
    uiParameterGruppe : UINT;
END_VAR
    Image (145,122 150x30), image: ImagePool.Kreis
    Frame (360,0 40x300)
        shows VIS_ANTRIEB_PARAMETER_LISTE(uiParameterGruppe := uiParameterGruppe)
    Frame (0,0 360x400), frame switch variable: uiParameterGruppe
        shows VIS_ANTRIEB_PARAMETER_BASE(ITF_ANTRIEBIN := ITF_ANTRIEBIN)
        shows VIS_ANTRIEB_PARAMETER_FUSES(ITF_ANTRIEBIN := ITF_ANTRIEBIN)
        shows VIS_ANTRIEB_PARAMETER_IO(ITF_ANTRIEBIN := ITF_ANTRIEBIN)
        shows VIS_ANTRIEB_PARAMETER_DATA(ITF_ANTRIEBIN := ITF_ANTRIEBIN)
        shows VIS_ANTRIEB_PARAMETER_TRENDLOG(ITF_ANTRIEBIN := ITF_ANTRIEBIN)
        pReferences[0]: ITF_Parameter=ITF_Parameter
        pReferences[1]: ITF_Parameter=ITF_Parameter
        pReferences[2]: ITF_Parameter=ITF_Parameter
        pReferences[3]: ITF_Parameter=ITF_Parameter
        pReferences[4]: ITF_Parameter=ITF_Parameter
END_VISUALIZATION

// 40 Visualizations/POPUP/PARAMETER/VIS_ANTRIEB_PARAMETER_LISTE
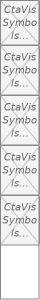
VISUALIZATION VIS_ANTRIEB_PARAMETER_LISTE  // 40x300
VAR_IN_OUT
	uiParameterGruppe : UINT;
END_VAR
    Rectangle (0,150 39x40), colour toggle: uiParameterGruppe = 3
        OnMouseDown: execute { uiParameterGruppe := 3; }
    Rectangle (0,100 39x40), colour toggle: uiParameterGruppe = 2
        OnMouseDown: execute { uiParameterGruppe := 2; }
    Rectangle (0,50 39x40), colour toggle: uiParameterGruppe = 1
        OnMouseDown: execute { uiParameterGruppe := 1; }
    Rectangle (0,0 39x40), colour toggle: uiParameterGruppe = 0
        OnMouseDown: execute { uiParameterGruppe := 0; }
    Image (0,0 40x45), image: CtaVisSymbols.ImagePool.engine
        OnMouseDown: execute { uiParameterGruppe := 0; }
    Image (0,45 40x50), image: CtaVisSymbols.ImagePool.lightning-bolt-circle
        OnMouseDown: execute { uiParameterGruppe := 1; }
    Image (0,95 40x50), image: CtaVisSymbols.ImagePool.dip-switch
        OnMouseDown: execute { uiParameterGruppe := 2; }
    Image (0,145 40x50), image: CtaVisSymbols.ImagePool.database_black
        OnMouseDown: execute { uiParameterGruppe := 3; }
    Rectangle (0,200 39x40), colour toggle: uiParameterGruppe = 4
        OnMouseDown: execute { uiParameterGruppe := 4; }
    Image (0,195 40x50), image: CtaVisSymbols.ImagePool.sine-wave
        OnMouseDown: execute { uiParameterGruppe := 4; }
END_VISUALIZATION

// 40 Visualizations/POPUP/MANUAL/VIS_ANTRIEB_MANUAL
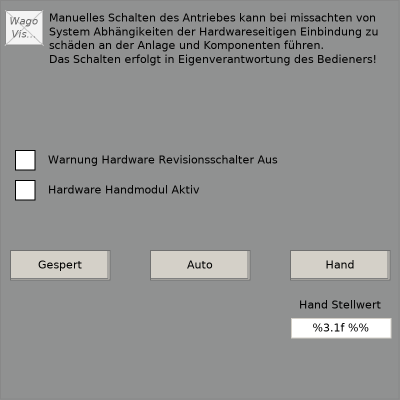
VISUALIZATION VIS_ANTRIEB_MANUAL  // 400x400
VAR_INPUT
    ITF_ANTRIEBIN    :   ITF_ANTRIEB;	
END_VAR
    Button (10,250 100x30), "Gespert", colour toggle: ITF_ANTRIEBIN.proHandOff, pressed state: ITF_ANTRIEBIN.proHandOff
        toggle ITF_ANTRIEBIN.proHandOff
    Button (290,250 100x30), "Hand", colour toggle: ITF_ANTRIEBIN.proHandOn, pressed state: ITF_ANTRIEBIN.proHandOn
        toggle ITF_ANTRIEBIN.proHandOn
    Button (150,250 100x30), "Auto", colour toggle: ITF_ANTRIEBIN.proAuto, pressed state: ITF_ANTRIEBIN.proAuto
        toggle ITF_ANTRIEBIN.proAuto
    Label (46,10 350x100), "Manuelles Schalten des Antriebes kann bei missachten von System Abhängikeiten der Hardwareseitigen Einbindung zu schäden an der Anlage und Komponenten führen. Das Schalten erfolgt in Eigenverantwortung des Bedieners!"
    Textfield (291,318 100x20), "%3.1f %%", text variable: ITF_ANTRIEBIN.proHandOnY, invisible if: NOT ITF_ANTRIEBIN.proIsRegulatet
        OnMouseClick: write the text variable via InputWithLimits, min 0, max 100, title 'Stellwert'
    Image (5,10 38x35), image: WagoVisuIcons.WagoIcons.2
    Label (290,295 100x20), "Hand Stellwert"
    Rectangle (15,180 20x20), colour toggle: ITF_ANTRIEBIN.proHardWareHandModulAktive, invisible if: NOT ITF_ANTRIEBIN.proHardWareHandModulAktive
    Label (45,180 200x20), "Hardware Handmodul Aktiv", invisible if: NOT ITF_ANTRIEBIN.proHardWareHandModulAktive
    Label (45,150 350x20), "Warnung Hardware Revisionsschalter Aus", invisible if: ITF_ANTRIEBIN.proRevisionSwitchOk
    Rectangle (15,150 20x20), colour toggle: NOT ITF_ANTRIEBIN.proRevisionSwitchOk, invisible if: ITF_ANTRIEBIN.proRevisionSwitchOk
END_VISUALIZATION

// 40 Visualizations/POPUP/OVERVIEW/VIS_ANTRIEB_OVERVIEW
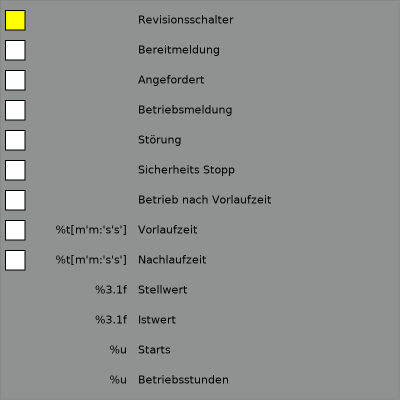
VISUALIZATION VIS_ANTRIEB_OVERVIEW  // 400x400
VAR_INPUT
    ITF_ANTRIEBIN    :   ITF_ANTRIEB;	
END_VAR
    Label (135,220 200x20), "Vorlaufzeit"
    Label (135,250 200x20), "Nachlaufzeit"
    Textfield (30,220 100x20), "%t[m'm:'s's']", text variable: ITF_ANTRIEBIN.proLeadTime
    Textfield (30,250 100x20), "%t[m'm:'s's']", text variable: ITF_ANTRIEBIN.proRunAfterTime
    Rectangle (5,220 20x20), colour toggle: ITF_ANTRIEBIN.proLeadTimeAktive
    Rectangle (5,250 20x20), colour toggle: ITF_ANTRIEBIN.proRunAfterTimeAktive
    Label (135,10 200x20), "Revisionsschalter"
    Label (135,40 200x20), "Bereitmeldung"
    Label (135,100 200x20), "Betriebsmeldung"
    Label (135,130 200x20), "Störung"
    Label (135,70 200x20), "Angefordert"
    Rectangle (5,10 20x20), colour toggle: ITF_ANTRIEBIN.proRevisionSwitchOk
    Rectangle (5,40 20x20), colour toggle: ITF_ANTRIEBIN.proIsReady
    Rectangle (5,70 20x20), colour toggle: ITF_ANTRIEBIN.proOn
    Rectangle (5,100 20x20), colour toggle: ITF_ANTRIEBIN.proMotorIsOn
    Rectangle (5,130 20x20), colour toggle: ITF_ANTRIEBIN.proIsError
    Label (135,160 200x20), "Sicherheits Stopp"
    Rectangle (5,160 20x20)
    Label (135,190 200x20), "Betrieb nach Vorlaufzeit"
    Rectangle (5,190 20x20), colour toggle: ITF_ANTRIEBIN.proIsOn
    Label (135,280 200x20), "Stellwert", invisible if: NOT ITF_ANTRIEBIN.proIsRegulatet
    Label (135,310 200x20), "Istwert", invisible if: NOT ITF_ANTRIEBIN.proIsRegulatet
    Textfield (30,280 100x20), "%3.1f", text variable: ITF_ANTRIEBIN.proOnY, invisible if: NOT ITF_ANTRIEBIN.proIsRegulatet
    Textfield (30,310 100x20), "%3.1f", text variable: ITF_ANTRIEBIN.proIsOnY, invisible if: NOT ITF_ANTRIEBIN.proIsRegulatet
    Textfield (30,370 100x20), "%u", text variable: ITF_ANTRIEBIN.proCountedHours
    Textfield (30,340 100x20), "%u", text variable: ITF_ANTRIEBIN.proCountedStarts
    Label (135,340 200x20), "Starts"
    Label (135,370 200x20), "Betriebsstunden"
END_VISUALIZATION

// 40 Visualizations/POPUP/BUS/AT_BUS
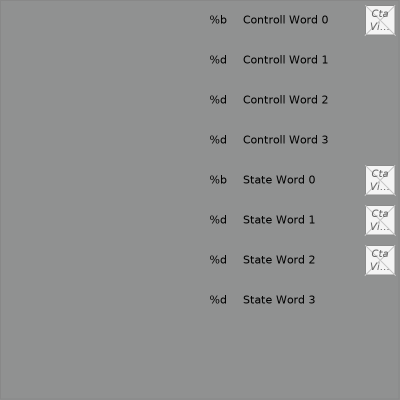
VISUALIZATION AT_BUS  // 400x400
VAR_INPUT
    ITF_ANTRIEBIN    :   ITF_ANTRIEB;	
END_VAR
    Frame (100,0 300x350)
        shows AT_BUS_CS(ITF_ANTRIEBIn := ITF_ANTRIEBIN, ayControllWord := ITF_ANTRIEBIN.proModbusControllWord, ayStateWord := ITF_ANTRIEBIN.proModbusStateWord)
END_VISUALIZATION

// 40 Visualizations/POPUP/BUS/AT_BUS_SW0_Detail
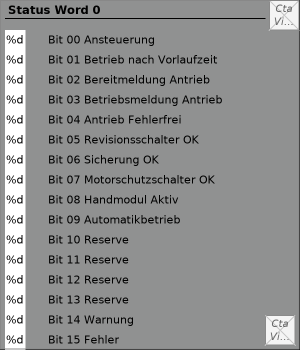
VISUALIZATION AT_BUS_SW0_Detail  // 300x350
VAR_IN_OUT
    wDetail     :   WORD;
END_VAR
VAR_INPUT	
    ITF_ANTRIEBIN    :   ITF_ANTRIEB;
END_VAR
VAR_IN_OUT
    xShow       :   BOOL;
END_VAR
    Rectangle (0,0 300x350)
    Textfield (5,30 20x20), "%d", text variable: TO_WORD(wDetail.0), input disabled if: NOT ITF_ANTRIEBIn.proModbusTest
        OnMouseClick: execute { wDetail.0 := NOT wDetail.0; }
    Label (45,30 220x20), "Bit 00 Ansteuerung"
    Textfield (5,50 20x20), "%d", text variable: TO_WORD(wDetail.1), input disabled if: NOT ITF_ANTRIEBIn.proModbusTest
        OnMouseClick: execute { wDetail.1 := NOT wDetail.1; }
    Label (45,50 220x20), "Bit 01 Betrieb nach Vorlaufzeit"
    Textfield (5,70 20x20), "%d", text variable: TO_WORD(wDetail.2), input disabled if: NOT ITF_ANTRIEBIn.proModbusTest
        OnMouseClick: execute { wDetail.2 := NOT wDetail.2; }
    Label (45,70 220x20), "Bit 02 Bereitmeldung Antrieb"
    Textfield (5,90 20x20), "%d", text variable: TO_WORD(wDetail.3), input disabled if: NOT ITF_ANTRIEBIn.proModbusTest
        OnMouseClick: execute { wDetail.3 := NOT wDetail.3; }
    Label (45,90 220x20), "Bit 03 Betriebsmeldung Antrieb"
    Textfield (5,110 20x20), "%d", text variable: TO_WORD(wDetail.4), input disabled if: NOT ITF_ANTRIEBIn.proModbusTest
        OnMouseClick: execute { wDetail.4 := NOT wDetail.4; }
    Label (45,110 220x20), "Bit 04 Antrieb Fehlerfrei"
    Textfield (5,130 20x20), "%d", text variable: TO_WORD(wDetail.5), input disabled if: NOT ITF_ANTRIEBIn.proModbusTest
        OnMouseClick: execute { wDetail.5 := NOT wDetail.5; }
    Label (45,130 220x20), "Bit 05 Revisionsschalter OK"
    Textfield (5,150 20x20), "%d", text variable: TO_WORD(wDetail.6), input disabled if: NOT ITF_ANTRIEBIn.proModbusTest
        OnMouseClick: execute { wDetail.6 := NOT wDetail.6; }
    Label (45,150 220x20), "Bit 06 Sicherung OK"
    Textfield (5,170 20x20), "%d", text variable: TO_WORD(wDetail.7), input disabled if: NOT ITF_ANTRIEBIn.proModbusTest
        OnMouseClick: execute { wDetail.7 := NOT wDetail.7; }
    Label (45,170 220x20), "Bit 07 Motorschutzschalter OK"
    Textfield (5,190 20x20), "%d", text variable: TO_WORD(wDetail.8), input disabled if: NOT ITF_ANTRIEBIn.proModbusTest
        OnMouseClick: execute { wDetail.8 := NOT wDetail.8; }
    Label (45,190 220x20), "Bit 08 Handmodul Aktiv"
    Textfield (5,210 20x20), "%d", text variable: TO_WORD(wDetail.9), input disabled if: NOT ITF_ANTRIEBIn.proModbusTest
        OnMouseClick: execute { wDetail.9 := NOT wDetail.9; }
    Label (45,210 220x20), "Bit 09 Automatikbetrieb"
    Textfield (5,230 20x20), "%d", text variable: TO_WORD(wDetail.10), input disabled if: NOT ITF_ANTRIEBIn.proModbusTest
        OnMouseClick: execute { wDetail.10 := NOT wDetail.10; }
    Label (45,230 220x20), "Bit 10 Reserve"
    Textfield (5,250 20x20), "%d", text variable: TO_WORD(wDetail.11), input disabled if: NOT ITF_ANTRIEBIn.proModbusTest
        OnMouseClick: execute { wDetail.11 := NOT wDetail.11; }
    Label (45,250 220x20), "Bit 11 Reserve"
    Textfield (5,270 20x20), "%d", text variable: TO_WORD(wDetail.12), input disabled if: NOT ITF_ANTRIEBIn.proModbusTest
        OnMouseClick: execute { wDetail.12 := NOT wDetail.12; }
    Label (45,270 220x20), "Bit 12 Reserve"
    Textfield (5,290 20x20), "%d", text variable: TO_WORD(wDetail.13), input disabled if: NOT ITF_ANTRIEBIn.proModbusTest
        OnMouseClick: execute { wDetail.13 := NOT wDetail.13; }
    Label (45,290 220x20), "Bit 13 Reserve"
    Textfield (5,310 20x20), "%d", text variable: TO_WORD(wDetail.14), input disabled if: NOT ITF_ANTRIEBIn.proModbusTest
        OnMouseClick: execute { wDetail.14 := NOT wDetail.14; }
    Label (45,310 220x20), "Bit 14 Warnung"
    Textfield (5,330 20x20), "%d", text variable: TO_WORD(wDetail.15), input disabled if: NOT ITF_ANTRIEBIn.proModbusTest
        OnMouseClick: execute { wDetail.15 := NOT wDetail.15; }
    Label (45,330 220x20), "Bit 15 Fehler"
    Image (269,0 30x30), image: CtaVisSymbols.ImagePool.close_solo_black
        OnMouseClick: execute { xShow := FALSE; ITF_ANTRIEBIN.proModbusTest := FALSE; }
    Label (5,0 150x20), "Status Word 0"
    Image (265,315 30x30), invisible if: ITF_ANTRIEBIN.proModbusTest, image: CtaVisSymbols.ImagePool.front_hand_Black
        OnMouseClick: execute { ITF_ANTRIEBIN.proModbusTest := TRUE; }
    Image (265,315 30x30), invisible if: NOT ITF_ANTRIEBIN.proModbusTest, image: CtaVisSymbols.ImagePool.front_hand_Yellow
        OnMouseClick: execute { ITF_ANTRIEBIN.proModbusTest := False; }
    Line (5,18) (265,18)
END_VISUALIZATION

// 40 Visualizations/POPUP/BUS/AT_BUS_CW0_Detail
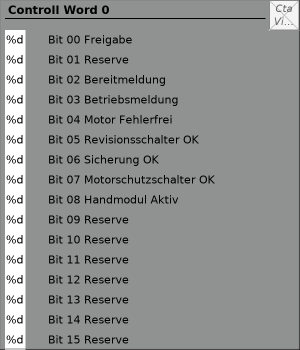
VISUALIZATION AT_BUS_CW0_Detail  // 300x350
VAR_IN_OUT
    wDetail :   WORD;
END_VAR
VAR_IN_OUT
    xShow   :   BOOL;
END_VAR
    Rectangle (0,0 300x350)
    Textfield (5,30 20x20), "%d", text variable: TO_WORD(wDetail.0), input disabled if: TRUE
    Label (45,30 180x20), "Bit 00 Freigabe"
    Textfield (5,50 20x20), "%d", text variable: TO_WORD(wDetail.1), input disabled if: TRUE
    Label (45,50 180x20), "Bit 01 Reserve"
    Textfield (5,70 20x20), "%d", text variable: TO_WORD(wDetail.2), input disabled if: TRUE
    Label (45,70 180x20), "Bit 02 Bereitmeldung"
    Textfield (5,90 20x20), "%d", text variable: TO_WORD(wDetail.3), input disabled if: TRUE
    Label (45,90 180x20), "Bit 03 Betriebsmeldung"
    Textfield (5,110 20x20), "%d", text variable: TO_WORD(wDetail.4), input disabled if: TRUE
    Label (45,110 180x20), "Bit 04 Motor Fehlerfrei"
    Textfield (5,130 20x20), "%d", text variable: TO_WORD(wDetail.5), input disabled if: TRUE
    Label (45,130 180x20), "Bit 05 Revisionsschalter OK"
    Textfield (5,150 20x20), "%d", text variable: TO_WORD(wDetail.6), input disabled if: TRUE
    Label (45,150 180x20), "Bit 06 Sicherung OK"
    Textfield (5,170 20x20), "%d", text variable: TO_WORD(wDetail.7), input disabled if: TRUE
    Label (45,170 180x20), "Bit 07 Motorschutzschalter OK"
    Textfield (5,190 20x20), "%d", text variable: TO_WORD(wDetail.8), input disabled if: TRUE
    Label (45,190 180x20), "Bit 08 Handmodul Aktiv"
    Textfield (5,210 20x20), "%d", text variable: TO_WORD(wDetail.9), input disabled if: TRUE
    Label (45,210 180x20), "Bit 09 Reserve"
    Textfield (5,230 20x20), "%d", text variable: TO_WORD(wDetail.10), input disabled if: TRUE
    Label (45,230 180x20), "Bit 10 Reserve"
    Textfield (5,250 20x20), "%d", text variable: TO_WORD(wDetail.11), input disabled if: TRUE
    Label (45,250 180x20), "Bit 11 Reserve"
    Textfield (5,270 20x20), "%d", text variable: TO_WORD(wDetail.12), input disabled if: TRUE
    Label (45,270 180x20), "Bit 12 Reserve"
    Textfield (5,290 20x20), "%d", text variable: TO_WORD(wDetail.13), input disabled if: TRUE
    Label (45,290 180x20), "Bit 13 Reserve"
    Textfield (5,310 20x20), "%d", text variable: TO_WORD(wDetail.14), input disabled if: TRUE
    Label (45,310 180x20), "Bit 14 Reserve"
    Textfield (5,330 20x20), "%d", text variable: TO_WORD(wDetail.15), input disabled if: TRUE
    Label (45,330 180x20), "Bit 15 Reserve"
    Image (269,0 30x30), image: CtaVisSymbols.ImagePool.close_solo_black
        OnMouseClick: execute { xShow := FALSE; }
    Label (5,0 150x20), "Controll Word 0"
    Line (5,18) (265,18)
END_VISUALIZATION

// 40 Visualizations/POPUP/BUS/AT_BUS_CS
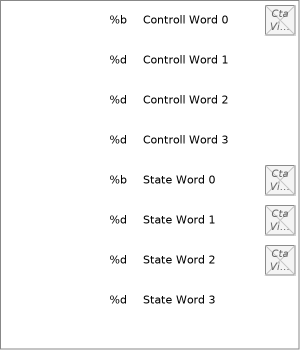
VISUALIZATION AT_BUS_CS  // 300x350
VAR_INPUT
    ITF_ANTRIEBIn        :   ITF_ANTRIEB;
    ayControllWord  :   REFERENCE TO ARRAY[0..3] OF WORD;
    ayStateWord     :   REFERENCE TO ARRAY[0..3] OF WORD;
END_VAR
VAR
    xShowCw :   BOOL;
    xShowSw :   BOOL;
    xShowSw1:   BOOL;
    xShowSw2:   BOOL;
END_VAR
    Textfield (0,10 130x20), "%b", text variable: ayControllWord[0]
    Label (140,10 120x20), "Controll Word 0"
    Label (140,50 120x20), "Controll Word 1"
    Textfield (0,50 130x20), "%d", text variable: ayControllWord[1]
    Label (140,90 120x20), "Controll Word 2", invisible if: TRUE
    Textfield (0,90 130x20), "%d", text variable: ayControllWord[2], invisible if: TRUE
    Label (140,130 120x20), "Controll Word 3", invisible if: TRUE
    Textfield (0,130 130x20), "%d", text variable: ayControllWord[2], invisible if: TRUE
    Image (265,5 30x30), image: CtaVisSymbols.ImagePool.information-variant
        OnMouseClick: execute {
            xShowCw := TRUE;
            xShowSw := FALSE;
            xShowSw1:= FALSE;
            xShowSw2:= FALSE;
        }
    Frame (300,0 300x350), invisible if: NOT xShowCw
        shows AT_BUS_CW0_Detail(wDetail := ayControllWord[0], xShow := xShowCw)
    Label (140,290 120x20), "State Word 3", invisible if: TRUE
    Textfield (0,170 130x20), "%b", text variable: ayStateWord[0]
        OnMouseDown: write the text variable via Default
    Label (140,170 120x20), "State Word 0"
    Label (140,210 120x20), "State Word 1"
    Textfield (0,210 130x20), "%d", text variable: ayStateWord[1]
    Label (140,250 120x20), "State Word 2"
    Textfield (0,250 130x20), "%d", text variable: ayStateWord[2]
    Textfield (0,290 130x20), "%d", text variable: ayStateWord[2], invisible if: TRUE
    Image (265,165 30x30), image: CtaVisSymbols.ImagePool.information-variant
        OnMouseClick: execute {
            xShowCw := FALSE;
            xShowSw := TRUE;
            xShowSw1:= FALSE;
            xShowSw2:= FALSE;
        }
    Frame (300,0 300x350), invisible if: NOT xShowSw
        shows AT_BUS_SW0_Detail(wDetail := ayStateWord[0], ITF_ANTRIEBIn := ITF_ANTRIEBIn, xShow := xShowSw)
        pReferences[0]: ITF_ATIn=ITF_ATIn
    Image (265,205 30x30), image: CtaVisSymbols.ImagePool.information-variant
        OnMouseClick: execute {
            xShowCw := FALSE;
            xShowSw := FALSE;
            xShowSw1:= TRUE;
            xShowSw2:= FALSE;
        }
    Frame (300,0 300x350), invisible if: NOT xShowSw1
        shows AT_BUS_SW1_Detail(wDetail := ayStateWord[1], ITF_ANTRIEBIn := ITF_ANTRIEBIn, xShow := xShowSw1)
    Frame (300,0 300x350), invisible if: NOT xShowSw2
        shows AT_BUS_SW2_Detail(wDetail := ayStateWord[2], ITF_ANTRIEBIn := ITF_ANTRIEBIn, xShow := xShowSw2)
    Image (265,245 30x30), image: CtaVisSymbols.ImagePool.information-variant
        OnMouseClick: execute {
            xShowCw := FALSE;
            xShowSw := FALSE;
            xShowSw1:= FALSE;
            xShowSw2:= TRUE;
        }
END_VISUALIZATION

// 40 Visualizations/POPUP/BUS/AT_BUS_SW1_Detail
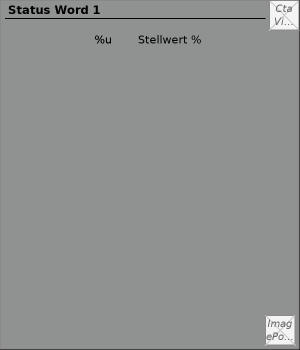
VISUALIZATION AT_BUS_SW1_Detail  // 300x350
VAR_IN_OUT
    wDetail     :   WORD;
END_VAR
VAR_INPUT	
    ITF_ANTRIEBIN    :   ITF_ANTRIEB;
END_VAR
VAR_IN_OUT
    xShow       :   BOOL;
END_VAR
    Rectangle (0,0 300x350)
    Image (269,0 30x30), image: CtaVisSymbols.ImagePool.close_solo_black
        OnMouseClick: execute { xShow := FALSE; ITF_ANTRIEBIN.proModbusTest := FALSE; }
    Label (5,0 150x20), "Status Word 1"
    Image (265,315 30x30), invisible if: ITF_ANTRIEBIN.proModbusTest, image: ImagePool.front_hand_FILL0_wght400_GRAD0_opsz48
        OnMouseClick: execute { ITF_ANTRIEBIN.proModbusTest := TRUE; }
    Image (265,315 30x30), invisible if: NOT ITF_ANTRIEBIn.proModbusTest, image: ImagePool.front_hand_FILL0_wght400_GRAD0_opsz48Yellow
        OnMouseClick: execute { ITF_ANTRIEBIN.proModbusTest := False; }
    Label (135,30 120x20), "Stellwert %"
    Textfield (5,30 110x20), "%u", text variable: wDetail, input disabled if: NOT ITF_ANTRIEBIn.proModbusTest
        OnMouseClick: write the text variable via InputWithLimits, min 0, max 100
    Textfield (5,30 110x20), "%u", text variable: wDetail, invisible if: ITF_ANTRIEBIN.proModbusTest
    Line (5,18) (265,18)
END_VISUALIZATION

// 40 Visualizations/POPUP/BUS/AT_BUS_SW2_Detail
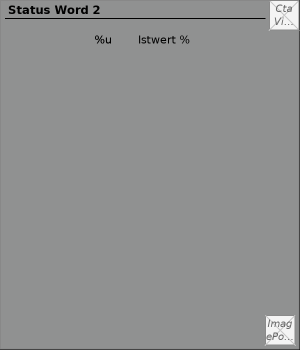
VISUALIZATION AT_BUS_SW2_Detail  // 300x350
VAR_IN_OUT
    wDetail             :   WORD;
END_VAR
VAR_INPUT	
    ITF_ANTRIEBIN       :   ITF_ANTRIEB;
END_VAR
VAR_IN_OUT
    xShow               :   BOOL;
END_VAR
    Rectangle (0,0 300x350)
    Image (269,0 30x30), image: CtaVisSymbols.ImagePool.close_solo_black
        OnMouseClick: execute { xShow := FALSE; ITF_ANTRIEBIN.proModbusTest := FALSE; }
    Label (5,0 150x20), "Status Word 2"
    Image (265,315 30x30), invisible if: ITF_ANTRIEBIn.proModbusTest, image: ImagePool.front_hand_FILL0_wght400_GRAD0_opsz48
        OnMouseClick: execute { ITF_ANTRIEBIN.proModbusTest := TRUE; }
    Image (265,315 30x30), invisible if: NOT ITF_ANTRIEBIN.proModbusTest, image: ImagePool.front_hand_FILL0_wght400_GRAD0_opsz48Yellow
        OnMouseClick: execute { ITF_ANTRIEBIN.proModbusTest := False; }
    Label (135,30 120x20), "Istwert %"
    Textfield (5,30 110x20), "%u", text variable: wDetail, input disabled if: NOT ITF_ANTRIEBIn.proModbusTest
        OnMouseClick: write the text variable via InputWithLimits, min 0, max 100
    Textfield (5,30 110x20), "%u", text variable: wDetail, invisible if: ITF_ANTRIEBIN.proModbusTest
    Line (5,18) (265,18)
END_VISUALIZATION

// 40 Visualizations/POPUP/REPORTS/VIS_ANTRIEB_REPORTS
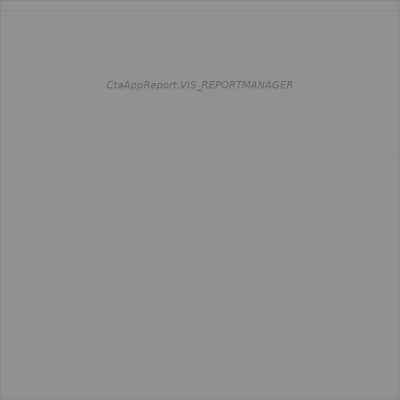
VISUALIZATION VIS_ANTRIEB_REPORTS  // 400x400
VAR_INPUT
    ITF_ANTRIEBIN    :   ITF_ANTRIEB;	
END_VAR
    Frame (0,10 400x150)
        shows CtaAppReport.VIS_REPORTMANAGER(ITF_REPORTMANAGER := ITF_ANTRIEBIN.proITF_REPORTMANAGER)
END_VISUALIZATION

// 40 Visualizations/POPUP/PARAMETER/AT_ParameterBase/VIS_ANTRIEB_PARAMETER_BASE0
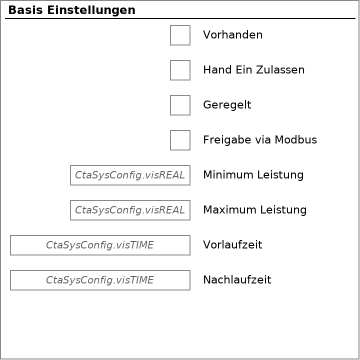
VISUALIZATION VIS_ANTRIEB_PARAMETER_BASE0  // 360x360
VAR_INPUT
    ITF_ANTRIEBIN    :   ITF_ANTRIEB;	
END_VAR
    Label (5,0 350x20), "Basis Einstellungen"
    Line (5,18) (355,18)
    Frame (170,25 20x20)
        shows CtaSysConfig.visBOOL(visfbBOOLIn := ITF_ANTRIEBIN.P_scBase_fbxEnable)
    Label (200,25 150x20), "Vorhanden"
    Frame (170,95 20x20)
        shows CtaSysConfig.visBOOL(visfbBOOLIn := ITF_ANTRIEBIN.P_scBase_fbxRegulatet)
    Label (200,95 150x20), "Geregelt"
    Frame (170,130 20x20)
        shows CtaSysConfig.visBOOL(visfbBOOLIn := ITF_ANTRIEBIN.P_scBase_fbxControllMb)
    Label (200,130 150x20), "Freigabe via Modbus"
    Frame (70,165 120x20)
        shows CtaSysConfig.visREAL(visfbREALIn := ITF_ANTRIEBIN.P_scBase_fbrYMin, stPhysikalischeEinheit := '%')
    Label (200,165 150x20), "Minimum Leistung"
    Frame (70,200 120x20)
        shows CtaSysConfig.visREAL(visfbREALIn := ITF_ANTRIEBIN.P_scBase_fbrYMax, stPhysikalischeEinheit := '%')
    Label (200,200 150x20), "Maximum Leistung"
    Frame (10,235 180x20)
        shows CtaSysConfig.visTIME(visfbTIMEIn := ITF_ANTRIEBIN.P_scBase_fbtLeadTime)
    Label (200,235 150x20), "Vorlaufzeit"
    Label (200,270 150x20), "Nachlaufzeit"
    Frame (10,270 180x20)
        shows CtaSysConfig.visTIME(visfbTIMEIn := ITF_ANTRIEBIN.P_scBase_fbtRunAfterTime)
    Frame (170,60 20x20)
        shows CtaSysConfig.visBOOL(visfbBOOLIn := ITF_ANTRIEBIN.P_scManual_fbxAlowManualOn)
    Label (200,60 150x20), "Hand Ein Zulassen"
END_VISUALIZATION

// 40 Visualizations/POPUP/PARAMETER/AT_ParameterBase/VIS_ANTRIEB_PARAMETER_BASE
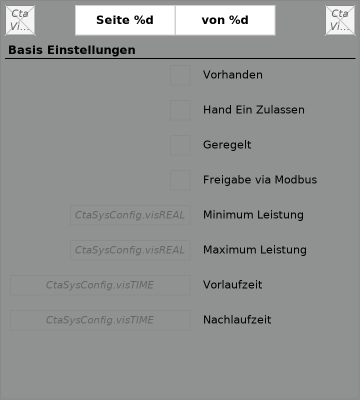
VISUALIZATION VIS_ANTRIEB_PARAMETER_BASE  // 360x400
VAR_INPUT
    ITF_ANTRIEBIN    :   ITF_ANTRIEB;	
END_VAR
VAR
    uiPage  :   UINT;
    uiMin   :   UINT    := 0;
    uiMax   :   UINT    := 0;
END_VAR
    Image (5,5 30x30), invisible if: uiPage = uiMin, image: CtaVisSymbols.ImagePool.arrow-left_square
        OnMouseClick: execute {
            uiPage := uiPage - 1;
            IF uiPage <= uiMin THEN
                uiPage := uiMin;
            END_IF;
        }
    Image (325,5 30x30), invisible if: uiPage = uiMax, image: CtaVisSymbols.ImagePool.arrow-right_square
        OnMouseClick: execute {
            uiPage := uiPage + 1;
            IF uiPage >= uiMax THEN
                uiPage := uiMax;
            END_IF;
        }
    Frame (0,40 360x360), frame switch variable: uiPage
        shows VIS_ANTRIEB_PARAMETER_BASE0(ITF_ANTRIEBIN := ITF_ANTRIEBIN)
        shows AT_ParameterIO1(ITF_Parameter := ITF_Parameter)
        pReferences[0]: ITF_Parameter=ITF_Parameter
    Textfield (175,5 100x30), "von %d", text variable: uiMax
    Textfield (75,5 100x30), "Seite %d", text variable: uiPage
END_VISUALIZATION

// 40 Visualizations/POPUP/PARAMETER/AT_Data/VIS_ANTRIEB_PARAMETER_DATA0
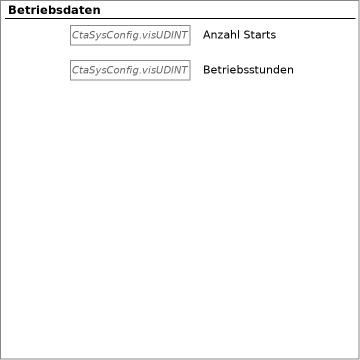
VISUALIZATION VIS_ANTRIEB_PARAMETER_DATA0  // 360x360
VAR_INPUT
    ITF_ANTRIEBIN    :   ITF_ANTRIEB;	
END_VAR
    Label (200,25 150x20), "Anzahl Starts"
    Label (200,60 150x20), "Betriebsstunden"
    Label (5,0 350x20), "Betriebsdaten"
    Frame (70,25 120x20)
        shows CtaSysConfig.visUDINT(visfbUDINTIn := ITF_ANTRIEBIN.P_scData_fbudiOperationStarts)
    Frame (70,60 120x20)
        shows CtaSysConfig.visUDINT(visfbUDINTIn := ITF_ANTRIEBIN.P_scData_fbudiOperatingHours)
    Line (5,18) (355,18)
END_VISUALIZATION

// 40 Visualizations/POPUP/PARAMETER/AT_Data/VIS_ANTRIEB_PARAMETER_DATA
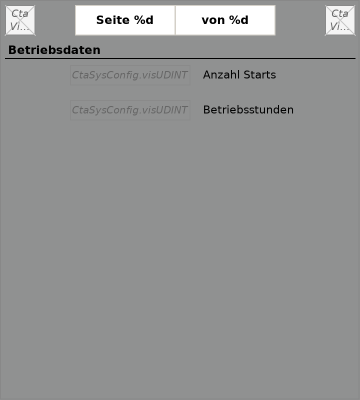
VISUALIZATION VIS_ANTRIEB_PARAMETER_DATA  // 360x400
VAR_INPUT
    ITF_ANTRIEBIN    :   ITF_ANTRIEB;	
END_VAR
VAR
    uiPage  :   UINT;
    uiMin   :   UINT    := 0;
    uiMax   :   UINT    := 0;
END_VAR
    Image (5,5 30x30), invisible if: uiPage = uiMin, image: CtaVisSymbols.ImagePool.arrow-left_square
        OnMouseClick: execute {
            uiPage := uiPage - 1;
            IF uiPage <= uiMin THEN
                uiPage := uiMin;
            END_IF;
        }
    Image (325,5 30x30), invisible if: uiPage = uiMax, image: CtaVisSymbols.ImagePool.arrow-right_square
        OnMouseClick: execute {
            uiPage := uiPage + 1;
            IF uiPage >= uiMax THEN
                uiPage := uiMax;
            END_IF;
        }
    Frame (0,40 360x360), frame switch variable: uiPage
        shows VIS_ANTRIEB_PARAMETER_DATA0(ITF_ANTRIEBIN := ITF_ANTRIEBIN)
        shows AT_ParameterIO1(ITF_Parameter := ITF_Parameter)
        pReferences[0]: ITF_Parameter=ITF_Parameter
    Textfield (75,5 100x30), "Seite %d", text variable: uiPage
    Textfield (175,5 100x30), "von %d", text variable: uiMax
END_VISUALIZATION

// 40 Visualizations/POPUP/PARAMETER/AT_Fuse/VIS_ANTRIEB_PARAMETER_FUSES0
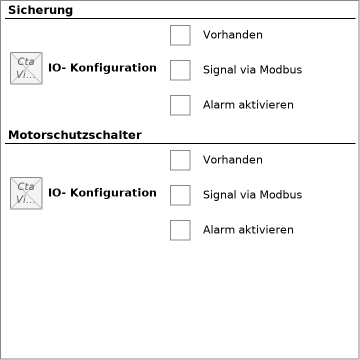
VISUALIZATION VIS_ANTRIEB_PARAMETER_FUSES0  // 360x360
VAR_INPUT
    ITF_ANTRIEBIN  		:	ITF_ANTRIEB;
	ITF_Fuse_IN			:	CtaSysIO.ITF_IO;
	ITF_MotorFuse_IN	:	CtaSysIO.ITF_IO;
END_VAR
    Frame (170,25 20x20)
        shows CtaSysConfig.visBOOL(visfbBOOLIn := ITF_ANTRIEBIN.P_scFuse_fbxEnable)
    Label (200,25 150x20), "Vorhanden"
    Frame (170,60 20x20)
        shows CtaSysConfig.visBOOL(visfbBOOLIn := ITF_ANTRIEBIN.P_scFuse_fbxInputMb)
    Label (200,60 150x20), "Signal via Modbus"
    Frame (170,95 20x20)
        shows CtaSysConfig.visBOOL(visfbBOOLIn := ITF_ANTRIEBIN.P_scFuse_fbxDoesAlarm)
    Label (200,95 150x20), "Alarm aktivieren"
    Label (5,0 350x20), "Sicherung"
    Label (5,125 350x20), "Motorschutzschalter"
    Frame (170,150 20x20)
        shows CtaSysConfig.visBOOL(visfbBOOLIn := ITF_ANTRIEBIN.P_scMotorFuse_fbxEnable)
    Label (200,150 150x20), "Vorhanden"
    Frame (170,185 20x20)
        shows CtaSysConfig.visBOOL(visfbBOOLIn := ITF_ANTRIEBIN.P_scMotorFuse_fbxInputMb)
    Label (200,185 150x20), "Signal via Modbus"
    Frame (170,220 20x20)
        shows CtaSysConfig.visBOOL(visfbBOOLIn := ITF_ANTRIEBIN.P_scMotorFuse_fbxDoesAlarm)
    Label (200,220 150x20), "Alarm aktivieren"
    Line (5,18) (355,18)
    Line (5,143) (355,143)
    Image (10,52 32x32), invisible if: ITF_Fuse_IN = 0, image: CtaVisSymbols.ImagePool.build
        OnMouseDown:  Dialog=VIS_ANTRIEB_POPUP_IO_ITF, Parameters={ITF_IO_IN: ITF_Fuse_IN}, OpenModal=True, OpenCentered=True
    Image (10,177 32x32), invisible if: ITF_MotorFuse_IN = 0, image: CtaVisSymbols.ImagePool.build
        OnMouseDown:  Dialog=VIS_ANTRIEB_POPUP_IO_ITF, Parameters={ITF_IO_IN: ITF_MotorFuse_IN}, OpenModal=True, OpenCentered=True
    Label (45,58 120x20), "IO- Konfiguration", invisible if: ITF_Fuse_IN = 0
    Label (45,183 120x20), "IO- Konfiguration", invisible if: ITF_MotorFuse_IN = 0
END_VISUALIZATION

// 40 Visualizations/POPUP/PARAMETER/AT_Fuse/VIS_ANTRIEB_PARAMETER_FUSES
